(* Schneider Machine Expert - Basic project FlandersHVL, file version 1.8.0.0 *)
(* ProjectInformations: Name=New project *)

HARDWARE
  Cpu 0: TM221CE24R
  ModuleExtensionObject 0: TM3AQ4/G
  ModuleExtensionObject 1: TM2DDO8TT
  ModuleExtensionObject 2: TM2DDO8TT
  EthernetConfiguration: NetworkName=M221, IpAllocationMode=FixedAddress, IpAddress=192.168.1.11, SubnetMask=255.255.255.0
  SerialLineConfiguration: Baud=Baud19200, Parity=ParityEven, DataBits=DataBits8, StopBits=StopBits1, PhysicalMedium=PhysicalMediumRs485, TransmissionMode=TransmissionModeModbusRtu, SlaveId=1, Addressing=SlaveAddressing
  MastTask: UsePeriodScanMode=false, PeriodScan=100
  FastTask: Period=255
  CpuBehavior: StartingMode=StartAsPreviousState, AutoSaveRamOnEeprom=true, WatchdogPeriod=250

SYMBOLS  (address, symbol, comment, settings)
  %M0       STOP
  %M1       RUN_STRIP_PULL_CYCLE
  %M2       EXTEND_CLAMP
  %M3       GLUE_TIMER_DN
  %M4       RUN_GLUE_CYCLE
  %M5       SYSTEM_RUNNING
  %M6       MCR  "Master Control Relay"
  %M7       SYSTEM_IDLE
  %M8       SYSTEM_START
  %M9       PHYSICAL_ALARM_TIMEOUT
  %M10      SYNC_STRIPS
  %M11      ONE_MIN_PASSED
  %M12      NEXT_SPEED
  %M13      START_RPM_TEST
  %M14      STRIP_PULL_STEP_1
  %M15      STRIP_PULL_LAST_STEP
  %M16      SYNC_VACS
  %M17      SYNC_STRIP_CYL_OUT
  %M18      SYN_STRIP_CYL_IN
  %M19      SYNC_PINS
  %M20      SYNC_GLUE
  %M21      SYNC_STRIP_MOTORS
  %M22      TEST_GLUE_RUNNING
  %M23      SLOW_JOG
  %M24      RUN_STRIP_PULL_A_CYCLE
  %M25      STRIP_PULL_A_MANUAL
  %M26      STRIP_PULL_B_MANUAL
  %M27      RUN_STRIP_PULL_B_CYCLE
  %M100     TEST_BIT
  %MW4      DRIVE_MOTOR_SETPOINT
  %MW5      MEDIA_DETECT_SETPOINT
  %MW6      GLUE_A_TOP_ON_DELAY_SETPOINT
  %MW7      VAC_ON_DELAY_SETPOINT
  %MW8      VAC_OFF_DELAY_SETPOINT
  %MW9      PIN_TIMER_SETPOINT
  %MW10     GLUE_A_TOP_OFF_DELAY_SETPOINT
  %MW11     GLUE_A_BOT_ON_DELAY_SETPOINT
  %MW12     GLUE_A_BOT_OFF_DELAY_SETPOINT
  %MW13     GLUE_B_TOP_ON_DELAY_SETPOINT
  %MW14     GLUE_B_TOP_OFF_DELAY_SETPOINT
  %MW15     GLUE_B_BOT_ON_DELAY_SETPOINT
  %MW16     GLUE_B_BOT_OFF_DELAY_SETPOINT
  %MF2      FILTERS_PER_MINUTE
  %TM0      GLUE_A_TOP_ON_DELAY  [Preset=200, Base=TenMilliSeconds]
  %TM1      GLUE_A_TOP_OFF_DELAY  [Preset=70, Base=TenMilliSeconds]
  %TM2      FPM_SPEED_TIMER  [Base=TenMilliSeconds]
  %TM3      MEDIA_DETECT_A_TIMER  [Preset=2000, Base=OneMilliSeconds]
  %TM4      VAC_A_ON_DELAY  [Preset=200, Base=OneMilliSeconds]
  %TM5      VAC_A_OFF_DELAY  [Preset=100, Base=OneMilliSeconds]
  %TM6      PIN_TIMER  [Preset=2, Base=TenMilliSeconds]
  %TM7      GLUE_A_BOT_ON_DELAY  [Base=TenMilliSeconds]
  %TM8      GLUE_A_BOT_OFF_DELAY  [Base=TenMilliSeconds]
  %TM9      GLUE_B_TOP_ON_DELAY  [Base=TenMilliSeconds]
  %TM10     GLUE_B_TOP_OFF_DELAY  [Base=TenMilliSeconds]
  %TM11     GLUE_B_BOT_ON_DELAY  [Base=TenMilliSeconds]
  %TM12     GLUE_B_BOT_OFF_DELAY  [Base=TenMilliSeconds]
  %TM13     VAC_B_ON_DELAY
  %TM14     VAC_B_OFF_DELAY
  %TM15     MEDIA_DETECT_B_TIMER
  %C0       FILTER_PER_MINUTE_COUNTER
  %I0.0     SPEED_DETECT
  %I0.1     FLIGHT_DETECT
  %I0.2     STRIP_CYL_A_OUT
  %I0.3     STRIP_CYL_A_IN
  %I0.4     STRIP_CYL_B_OUT
  %I0.5     STRIP_CYL_B_IN
  %I0.6     MEDIA_DETECT
  %I0.7     STRIP_DETECT_A
  %I0.8     STRIP_DETECT_B
  %I0.9     GLUE_EYE
  %I0.10    SAFETY
  %Q0.0     VAC_A
  %Q0.1     VAC_B
  %Q0.2     STRIP_ARM_A
  %Q0.3     STRIP_ARM_B
  %Q0.4     PIN_A
  %Q0.5     PIN_B
  %Q0.6     GLUE_HEAD_A_TOP
  %Q0.7     GLUE_HEAD_A_BOT
  %Q0.8     GLUE_HEAD_B_TOP
  %Q0.9     GLUE_HEAD_B_BOT
  %QW1.0    DRIVE_MOTOR  [Type=Type_0_10V, Scope=Scope_Customized, Minimum=0, Maximum=7000]
  %Q2.0     PHYSICAL_ALARM
  %Q2.3     PINCH_ROLLER_MOTOR
  %Q2.4     STRIP_B_MOTOR
  %Q2.5     STRIP_A_MOTOR
  %Q2.7     DRIVE_MOTOR_RUN
  %Q3.0     PAD_CUT

POU Strip_Machine_A
  (* SectionNumber=1 *)

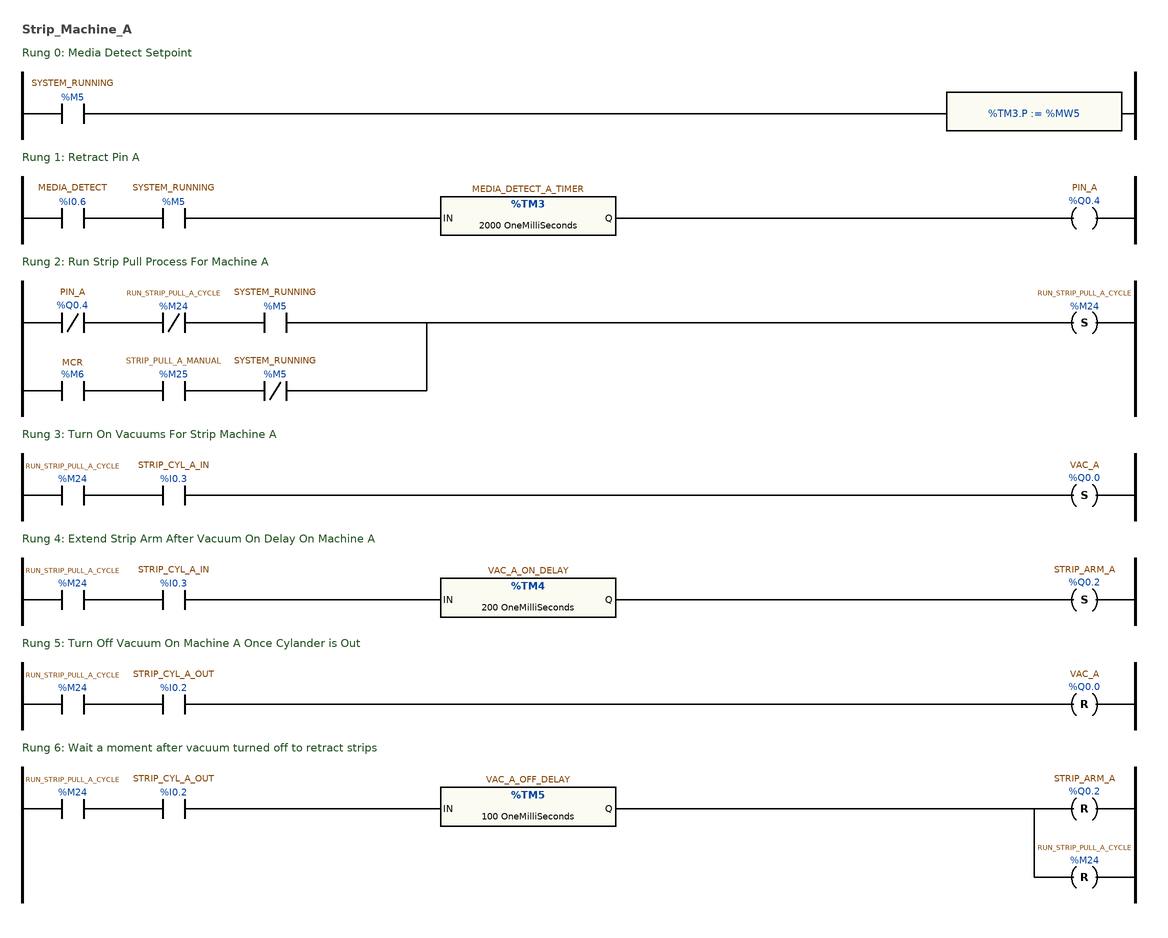

// Rung 0: Media Detect Setpoint
  LD %M5                  (* SYSTEM_RUNNING *)
  [ %TM3.P := %MW5 ]      (* MEDIA_DETECT_A_TIMER, MEDIA_DETECT_SETPOINT *)
  // as ST:
  //   IF SYSTEM_RUNNING THEN MEDIA_DETECT_A_TIMER.P := MEDIA_DETECT_SETPOINT; END_IF;

// Rung 1: Retract Pin A
  BLK %TM3                (* MEDIA_DETECT_A_TIMER *)
  LD %I0.6                (* MEDIA_DETECT *)
  AND %M5                 (* SYSTEM_RUNNING *)
  IN
  OUT_BLK
  LD Q
  ST %Q0.4                (* PIN_A *)
  END_BLK
  // as ST:
  //   MEDIA_DETECT_A_TIMER(IN := MEDIA_DETECT AND SYSTEM_RUNNING);
  //   PIN_A := MEDIA_DETECT_A_TIMER.Q;

// Rung 2: Run Strip Pull Process For Machine A
  LDN %Q0.4               (* PIN_A *)
  ANDN %M24               (* RUN_STRIP_PULL_A_CYCLE *)
  AND %M5                 (* SYSTEM_RUNNING *)
  OR( %M6                 (* MCR *)
  AND %M25                (* STRIP_PULL_A_MANUAL *)
  ANDN %M5                (* SYSTEM_RUNNING *)
  )
  S %M24                  (* RUN_STRIP_PULL_A_CYCLE *)
  // as ST:
  //   IF NOT PIN_A AND NOT RUN_STRIP_PULL_A_CYCLE AND SYSTEM_RUNNING OR MCR AND STRIP_PULL_A_MANUAL AND NOT SYSTEM_RUNNING THEN RUN_STRIP_PULL_A_CYCLE := TRUE; END_IF;

// Rung 3: Turn On Vacuums For Strip Machine A
  LD %M24                 (* RUN_STRIP_PULL_A_CYCLE *)
  AND %I0.3               (* STRIP_CYL_A_IN *)
  S %Q0.0                 (* VAC_A *)
  // as ST:
  //   IF RUN_STRIP_PULL_A_CYCLE AND STRIP_CYL_A_IN THEN VAC_A := TRUE; END_IF;

// Rung 4: Extend Strip Arm After Vacuum On Delay On Machine A
  BLK %TM4                (* VAC_A_ON_DELAY *)
  LD %M24                 (* RUN_STRIP_PULL_A_CYCLE *)
  AND %I0.3               (* STRIP_CYL_A_IN *)
  IN
  OUT_BLK
  LD Q
  S %Q0.2                 (* STRIP_ARM_A *)
  END_BLK
  // as ST:
  //   VAC_A_ON_DELAY(IN := RUN_STRIP_PULL_A_CYCLE AND STRIP_CYL_A_IN);
  //   IF VAC_A_ON_DELAY.Q THEN STRIP_ARM_A := TRUE; END_IF;

// Rung 5: Turn Off Vacuum On Machine A Once Cylander is Out
  LD %M24                 (* RUN_STRIP_PULL_A_CYCLE *)
  AND %I0.2               (* STRIP_CYL_A_OUT *)
  R %Q0.0                 (* VAC_A *)
  // as ST:
  //   IF RUN_STRIP_PULL_A_CYCLE AND STRIP_CYL_A_OUT THEN VAC_A := FALSE; END_IF;

// Rung 6: Wait a moment after vacuum turned off to retract strips
  BLK %TM5                (* VAC_A_OFF_DELAY *)
  LD %M24                 (* RUN_STRIP_PULL_A_CYCLE *)
  AND %I0.2               (* STRIP_CYL_A_OUT *)
  IN
  OUT_BLK
  LD Q
  R %Q0.2                 (* STRIP_ARM_A *)
  R %M24                  (* RUN_STRIP_PULL_A_CYCLE *)
  END_BLK
  // as ST:
  //   VAC_A_OFF_DELAY(IN := RUN_STRIP_PULL_A_CYCLE AND STRIP_CYL_A_OUT);
  //   IF VAC_A_OFF_DELAY.Q THEN STRIP_ARM_A := FALSE; END_IF;
  //   IF VAC_A_OFF_DELAY.Q THEN RUN_STRIP_PULL_A_CYCLE := FALSE; END_IF;

POU High_Power_Devices
  (* SectionNumber=2 *)

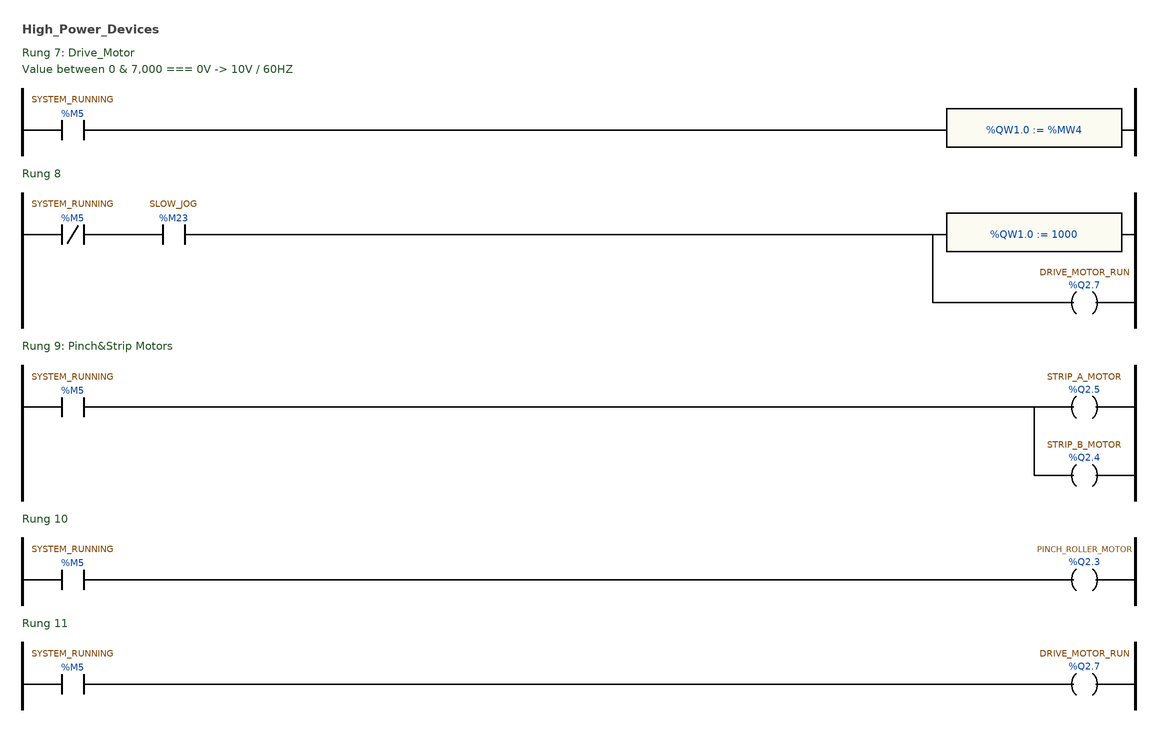

// Rung 7: Drive_Motor
// Value between 0 & 7,000 === 0V -> 10V / 60HZ
  LD %M5                  (* SYSTEM_RUNNING *)
  [ %QW1.0 := %MW4 ]      (* DRIVE_MOTOR, DRIVE_MOTOR_SETPOINT *)
  // as ST:
  //   IF SYSTEM_RUNNING THEN DRIVE_MOTOR := DRIVE_MOTOR_SETPOINT; END_IF;

// Rung 8
  LDN %M5                 (* SYSTEM_RUNNING *)
  AND %M23                (* SLOW_JOG *)
  [ %QW1.0 := 1000 ]      (* DRIVE_MOTOR *)
  ST %Q2.7                (* DRIVE_MOTOR_RUN *)
  // as ST:
  //   IF NOT SYSTEM_RUNNING AND SLOW_JOG THEN DRIVE_MOTOR := 1000; END_IF;
  //   DRIVE_MOTOR_RUN := NOT SYSTEM_RUNNING AND SLOW_JOG;

// Rung 9: Pinch&Strip Motors
  LD %M5                  (* SYSTEM_RUNNING *)
  ST %Q2.5                (* STRIP_A_MOTOR *)
  ST %Q2.4                (* STRIP_B_MOTOR *)
  // as ST:
  //   STRIP_A_MOTOR := SYSTEM_RUNNING;
  //   STRIP_B_MOTOR := SYSTEM_RUNNING;

// Rung 10
  LD %M5                  (* SYSTEM_RUNNING *)
  ST %Q2.3                (* PINCH_ROLLER_MOTOR *)
  // as ST:
  //   PINCH_ROLLER_MOTOR := SYSTEM_RUNNING;

// Rung 11
  LD %M5                  (* SYSTEM_RUNNING *)
  ST %Q2.7                (* DRIVE_MOTOR_RUN *)
  // as ST:
  //   DRIVE_MOTOR_RUN := SYSTEM_RUNNING;

POU RPM
  (* SectionNumber=3 *)

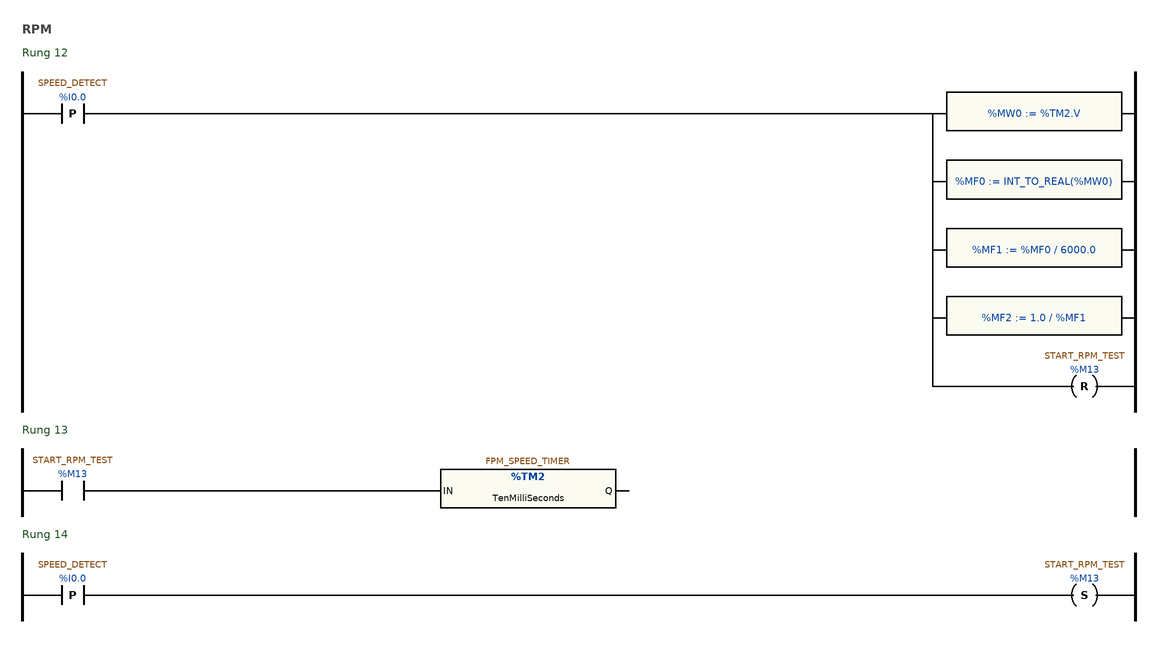

// Rung 12
  LDR %I0.0               (* SPEED_DETECT *)
  [ %MW0 := %TM2.V ]      (* FPM_SPEED_TIMER *)
  [ %MF0 := INT_TO_REAL ( %MW0 ) ]
  [ %MF1 := %MF0 / 6000.0 ]
  [ %MF2 := 1.0 / %MF1 ]  (* FILTERS_PER_MINUTE *)
  R %M13                  (* START_RPM_TEST *)
  // as ST:
  //   IF RISING(SPEED_DETECT) THEN %MW0 := FPM_SPEED_TIMER.V; END_IF;
  //   IF RISING(SPEED_DETECT) THEN %MF0 := INT_TO_REAL ( %MW0 ); END_IF;
  //   IF RISING(SPEED_DETECT) THEN %MF1 := %MF0  /  6000.0; END_IF;
  //   IF RISING(SPEED_DETECT) THEN FILTERS_PER_MINUTE := 1.0  /  %MF1; END_IF;
  //   IF RISING(SPEED_DETECT) THEN START_RPM_TEST := FALSE; END_IF;

// Rung 13
  BLK %TM2                (* FPM_SPEED_TIMER *)
  LD %M13                 (* START_RPM_TEST *)
  IN
  END_BLK
  // as ST:
  //   FPM_SPEED_TIMER(IN := START_RPM_TEST);

// Rung 14
  LDR %I0.0               (* SPEED_DETECT *)
  S %M13                  (* START_RPM_TEST *)
  // as ST:
  //   IF RISING(SPEED_DETECT) THEN START_RPM_TEST := TRUE; END_IF;

POU Synchronize
  (* SectionNumber=4 *)

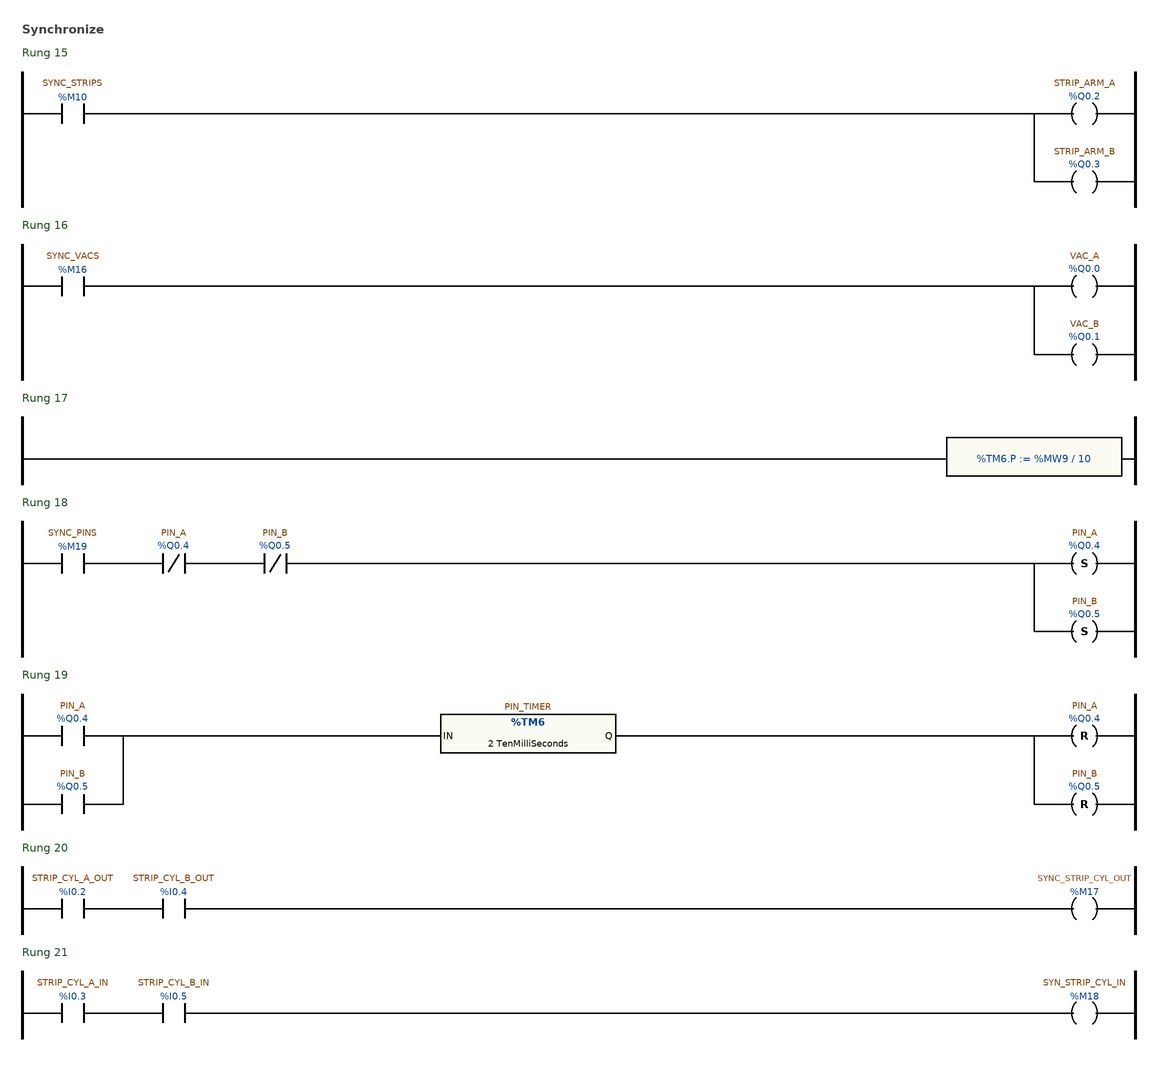

// Rung 15
  LD %M10                 (* SYNC_STRIPS *)
  ST %Q0.2                (* STRIP_ARM_A *)
  ST %Q0.3                (* STRIP_ARM_B *)
  // as ST:
  //   STRIP_ARM_A := SYNC_STRIPS;
  //   STRIP_ARM_B := SYNC_STRIPS;

// Rung 16
  LD %M16                 (* SYNC_VACS *)
  ST %Q0.0                (* VAC_A *)
  ST %Q0.1                (* VAC_B *)
  // as ST:
  //   VAC_A := SYNC_VACS;
  //   VAC_B := SYNC_VACS;

// Rung 17
  LD 1
  [ %TM6.P := %MW9 / 10 ] (* PIN_TIMER, PIN_TIMER_SETPOINT *)
  // as ST:
  //   PIN_TIMER.P := PIN_TIMER_SETPOINT / 10;

// Rung 18
  LD %M19                 (* SYNC_PINS *)
  ANDN %Q0.4              (* PIN_A *)
  ANDN %Q0.5              (* PIN_B *)
  S %Q0.4                 (* PIN_A *)
  S %Q0.5                 (* PIN_B *)
  // as ST:
  //   _t1 := SYNC_PINS AND NOT PIN_A AND NOT PIN_B;
  //   IF _t1 THEN PIN_A := TRUE; END_IF;
  //   IF _t1 THEN PIN_B := TRUE; END_IF;

// Rung 19
  BLK %TM6                (* PIN_TIMER *)
  LD %Q0.4                (* PIN_A *)
  OR %Q0.5                (* PIN_B *)
  IN
  OUT_BLK
  LD Q
  R %Q0.4                 (* PIN_A *)
  R %Q0.5                 (* PIN_B *)
  END_BLK
  // as ST:
  //   PIN_TIMER(IN := PIN_A OR PIN_B);
  //   IF PIN_TIMER.Q THEN PIN_A := FALSE; END_IF;
  //   IF PIN_TIMER.Q THEN PIN_B := FALSE; END_IF;

// Rung 20
  LD %I0.2                (* STRIP_CYL_A_OUT *)
  AND %I0.4               (* STRIP_CYL_B_OUT *)
  ST %M17                 (* SYNC_STRIP_CYL_OUT *)
  // as ST:
  //   SYNC_STRIP_CYL_OUT := STRIP_CYL_A_OUT AND STRIP_CYL_B_OUT;

// Rung 21
  LD %I0.3                (* STRIP_CYL_A_IN *)
  AND %I0.5               (* STRIP_CYL_B_IN *)
  ST %M18                 (* SYN_STRIP_CYL_IN *)
  // as ST:
  //   SYN_STRIP_CYL_IN := STRIP_CYL_A_IN AND STRIP_CYL_B_IN;

POU Sytem Signals
  (* SectionNumber=5 *)

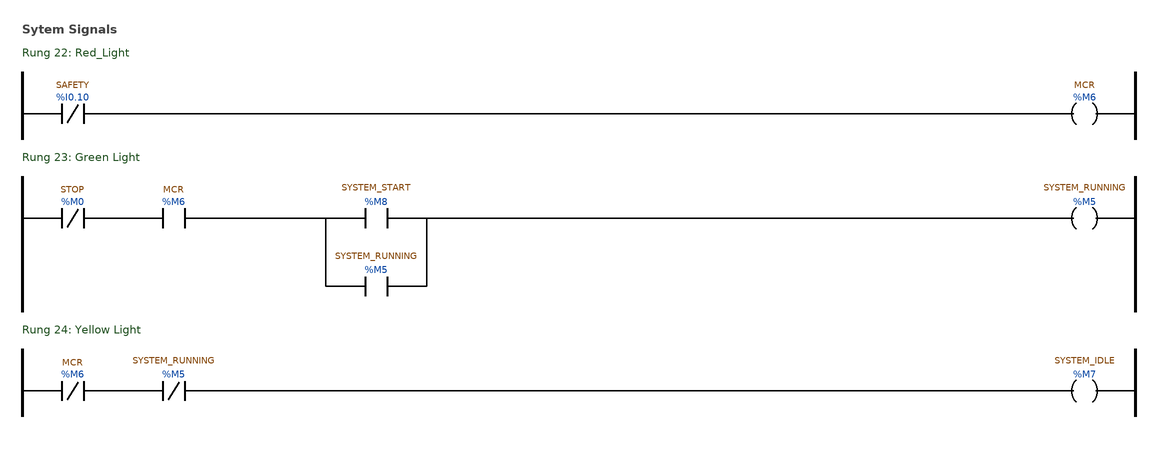

// Rung 22: Red_Light
  LDN %I0.10              (* SAFETY *)
  ST %M6                  (* MCR *)
  // as ST:
  //   MCR := NOT SAFETY;

// Rung 23: Green Light
  LDN %M0                 (* STOP *)
  AND %M6                 (* MCR *)
  AND( %M8                (* SYSTEM_START *)
  OR %M5                  (* SYSTEM_RUNNING *)
  )
  ST %M5                  (* SYSTEM_RUNNING *)
  // as ST:
  //   SYSTEM_RUNNING := NOT STOP AND MCR AND (SYSTEM_START OR SYSTEM_RUNNING);

// Rung 24: Yellow Light
  LDN %M6                 (* MCR *)
  ANDN %M5                (* SYSTEM_RUNNING *)
  ST %M7                  (* SYSTEM_IDLE *)
  // as ST:
  //   SYSTEM_IDLE := NOT MCR AND NOT SYSTEM_RUNNING;

POU Glue
  (* SectionNumber=6 *)

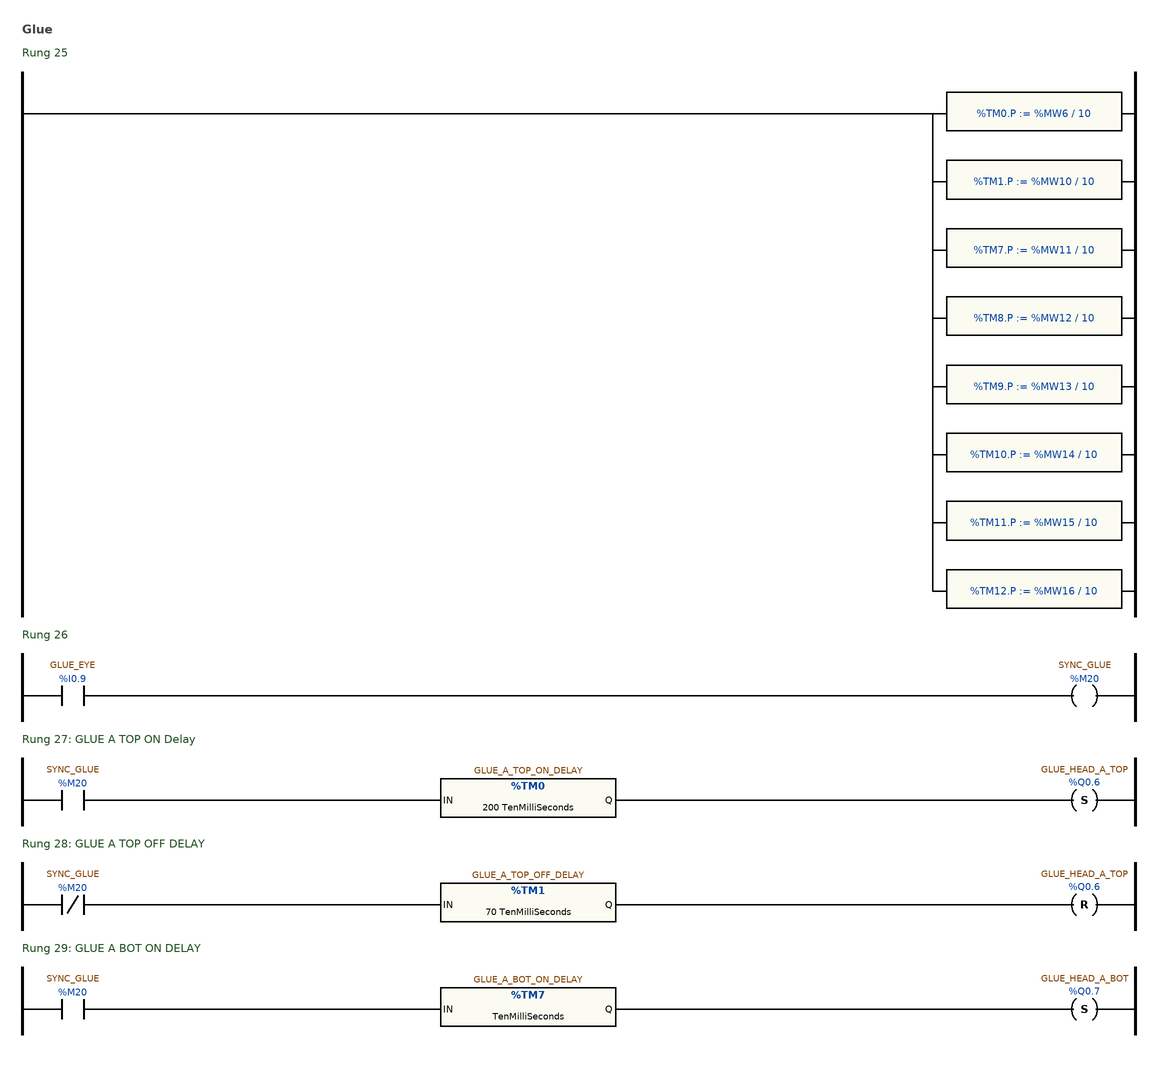

// Rung 25
  LD 1
  [%TM0.P := %MW6 / 10]   (* GLUE_A_TOP_ON_DELAY, GLUE_A_TOP_ON_DELAY_SETPOINT *)
  [%TM1.P := %MW10 / 10]  (* GLUE_A_TOP_OFF_DELAY, GLUE_A_TOP_OFF_DELAY_SETPOINT *)
  [%TM7.P := %MW11 / 10]  (* GLUE_A_BOT_ON_DELAY, GLUE_A_BOT_ON_DELAY_SETPOINT *)
  [%TM8.P := %MW12 / 10]  (* GLUE_A_BOT_OFF_DELAY, GLUE_A_BOT_OFF_DELAY_SETPOINT *)
  [%TM9.P := %MW13 / 10]  (* GLUE_B_TOP_ON_DELAY, GLUE_B_TOP_ON_DELAY_SETPOINT *)
  [%TM10.P := %MW14 / 10] (* GLUE_B_TOP_OFF_DELAY, GLUE_B_TOP_OFF_DELAY_SETPOINT *)
  [%TM11.P := %MW15 / 10] (* GLUE_B_BOT_ON_DELAY, GLUE_B_BOT_ON_DELAY_SETPOINT *)
  [%TM12.P := %MW16 / 10] (* GLUE_B_BOT_OFF_DELAY, GLUE_B_BOT_OFF_DELAY_SETPOINT *)
  // as ST:
  //   GLUE_A_TOP_ON_DELAY.P := GLUE_A_TOP_ON_DELAY_SETPOINT / 10;
  //   GLUE_A_TOP_OFF_DELAY.P := GLUE_A_TOP_OFF_DELAY_SETPOINT / 10;
  //   GLUE_A_BOT_ON_DELAY.P := GLUE_A_BOT_ON_DELAY_SETPOINT / 10;
  //   GLUE_A_BOT_OFF_DELAY.P := GLUE_A_BOT_OFF_DELAY_SETPOINT / 10;
  //   GLUE_B_TOP_ON_DELAY.P := GLUE_B_TOP_ON_DELAY_SETPOINT / 10;
  //   GLUE_B_TOP_OFF_DELAY.P := GLUE_B_TOP_OFF_DELAY_SETPOINT / 10;
  //   GLUE_B_BOT_ON_DELAY.P := GLUE_B_BOT_ON_DELAY_SETPOINT / 10;
  //   GLUE_B_BOT_OFF_DELAY.P := GLUE_B_BOT_OFF_DELAY_SETPOINT / 10;

// Rung 26
  LD %I0.9                (* GLUE_EYE *)
  ST %M20                 (* SYNC_GLUE *)
  // as ST:
  //   SYNC_GLUE := GLUE_EYE;

// Rung 27: GLUE A TOP ON Delay
  BLK %TM0                (* GLUE_A_TOP_ON_DELAY *)
  LD %M20                 (* SYNC_GLUE *)
  IN
  OUT_BLK
  LD Q
  S %Q0.6                 (* GLUE_HEAD_A_TOP *)
  END_BLK
  // as ST:
  //   GLUE_A_TOP_ON_DELAY(IN := SYNC_GLUE);
  //   IF GLUE_A_TOP_ON_DELAY.Q THEN GLUE_HEAD_A_TOP := TRUE; END_IF;

// Rung 28: GLUE A TOP OFF DELAY
  BLK %TM1                (* GLUE_A_TOP_OFF_DELAY *)
  LDN %M20                (* SYNC_GLUE *)
  IN
  OUT_BLK
  LD Q
  R %Q0.6                 (* GLUE_HEAD_A_TOP *)
  END_BLK
  // as ST:
  //   GLUE_A_TOP_OFF_DELAY(IN := NOT SYNC_GLUE);
  //   IF GLUE_A_TOP_OFF_DELAY.Q THEN GLUE_HEAD_A_TOP := FALSE; END_IF;

// Rung 29: GLUE A BOT ON DELAY
  BLK %TM7                (* GLUE_A_BOT_ON_DELAY *)
  LD %M20                 (* SYNC_GLUE *)
  IN
  OUT_BLK
  LD Q
  S %Q0.7                 (* GLUE_HEAD_A_BOT *)
  END_BLK
  // as ST:
  //   GLUE_A_BOT_ON_DELAY(IN := SYNC_GLUE);
  //   IF GLUE_A_BOT_ON_DELAY.Q THEN GLUE_HEAD_A_BOT := TRUE; END_IF;

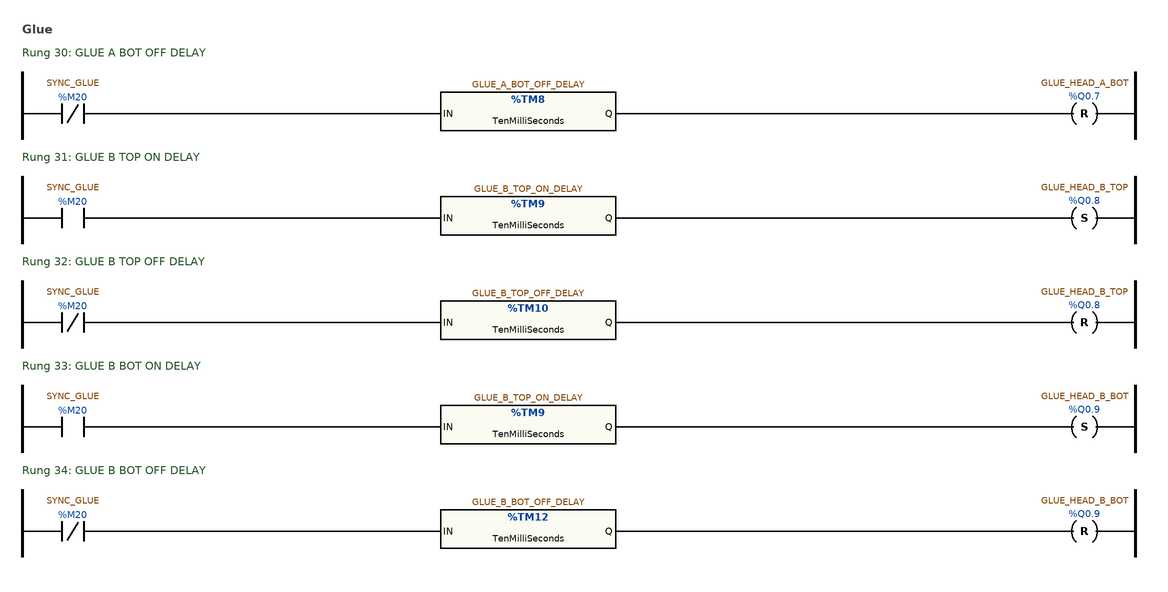

// Rung 30: GLUE A BOT OFF DELAY
  BLK %TM8                (* GLUE_A_BOT_OFF_DELAY *)
  LDN %M20                (* SYNC_GLUE *)
  IN
  OUT_BLK
  LD Q
  R %Q0.7                 (* GLUE_HEAD_A_BOT *)
  END_BLK
  // as ST:
  //   GLUE_A_BOT_OFF_DELAY(IN := NOT SYNC_GLUE);
  //   IF GLUE_A_BOT_OFF_DELAY.Q THEN GLUE_HEAD_A_BOT := FALSE; END_IF;

// Rung 31: GLUE B TOP ON DELAY
  BLK %TM9                (* GLUE_B_TOP_ON_DELAY *)
  LD %M20                 (* SYNC_GLUE *)
  IN
  OUT_BLK
  LD Q
  S %Q0.8                 (* GLUE_HEAD_B_TOP *)
  END_BLK
  // as ST:
  //   GLUE_B_TOP_ON_DELAY(IN := SYNC_GLUE);
  //   IF GLUE_B_TOP_ON_DELAY.Q THEN GLUE_HEAD_B_TOP := TRUE; END_IF;

// Rung 32: GLUE B TOP OFF DELAY
  BLK %TM10               (* GLUE_B_TOP_OFF_DELAY *)
  LDN %M20                (* SYNC_GLUE *)
  IN
  OUT_BLK
  LD Q
  R %Q0.8                 (* GLUE_HEAD_B_TOP *)
  END_BLK
  // as ST:
  //   GLUE_B_TOP_OFF_DELAY(IN := NOT SYNC_GLUE);
  //   IF GLUE_B_TOP_OFF_DELAY.Q THEN GLUE_HEAD_B_TOP := FALSE; END_IF;

// Rung 33: GLUE B BOT ON DELAY
  BLK %TM9                (* GLUE_B_TOP_ON_DELAY *)
  LD %M20                 (* SYNC_GLUE *)
  IN
  OUT_BLK
  LD Q
  S %Q0.9                 (* GLUE_HEAD_B_BOT *)
  END_BLK
  // as ST:
  //   GLUE_B_TOP_ON_DELAY(IN := SYNC_GLUE);
  //   IF GLUE_B_TOP_ON_DELAY.Q THEN GLUE_HEAD_B_BOT := TRUE; END_IF;

// Rung 34: GLUE B BOT OFF DELAY
  BLK %TM12               (* GLUE_B_BOT_OFF_DELAY *)
  LDN %M20                (* SYNC_GLUE *)
  IN
  OUT_BLK
  LD Q
  R %Q0.9                 (* GLUE_HEAD_B_BOT *)
  END_BLK
  // as ST:
  //   GLUE_B_BOT_OFF_DELAY(IN := NOT SYNC_GLUE);
  //   IF GLUE_B_BOT_OFF_DELAY.Q THEN GLUE_HEAD_B_BOT := FALSE; END_IF;

POU Timer_Setpoints
  (* SectionNumber=7 *)

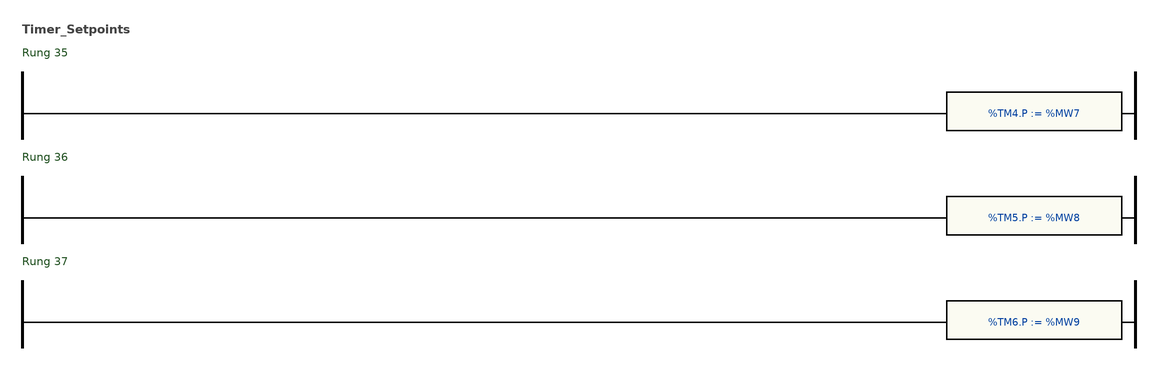

// Rung 35
  LD 1
  [ %TM4.P := %MW7 ]      (* VAC_A_ON_DELAY, VAC_ON_DELAY_SETPOINT *)
  // as ST:
  //   VAC_A_ON_DELAY.P := VAC_ON_DELAY_SETPOINT;

// Rung 36
  LD 1
  [ %TM5.P := %MW8 ]      (* VAC_A_OFF_DELAY, VAC_OFF_DELAY_SETPOINT *)
  // as ST:
  //   VAC_A_OFF_DELAY.P := VAC_OFF_DELAY_SETPOINT;

// Rung 37
  LD 1
  [ %TM6.P := %MW9 ]      (* PIN_TIMER, PIN_TIMER_SETPOINT *)
  // as ST:
  //   PIN_TIMER.P := PIN_TIMER_SETPOINT;

POU Pad Cutter
  (* SectionNumber=0 *)

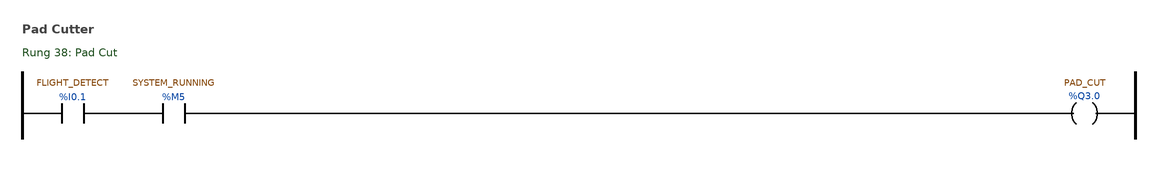

// Rung 38: Pad Cut
  LD %I0.1                (* FLIGHT_DETECT *)
  AND %M5                 (* SYSTEM_RUNNING *)
  ST %Q3.0                (* PAD_CUT *)
  // as ST:
  //   PAD_CUT := FLIGHT_DETECT AND SYSTEM_RUNNING;

POU Strip_Machine_B
  (* SectionNumber=1 *)

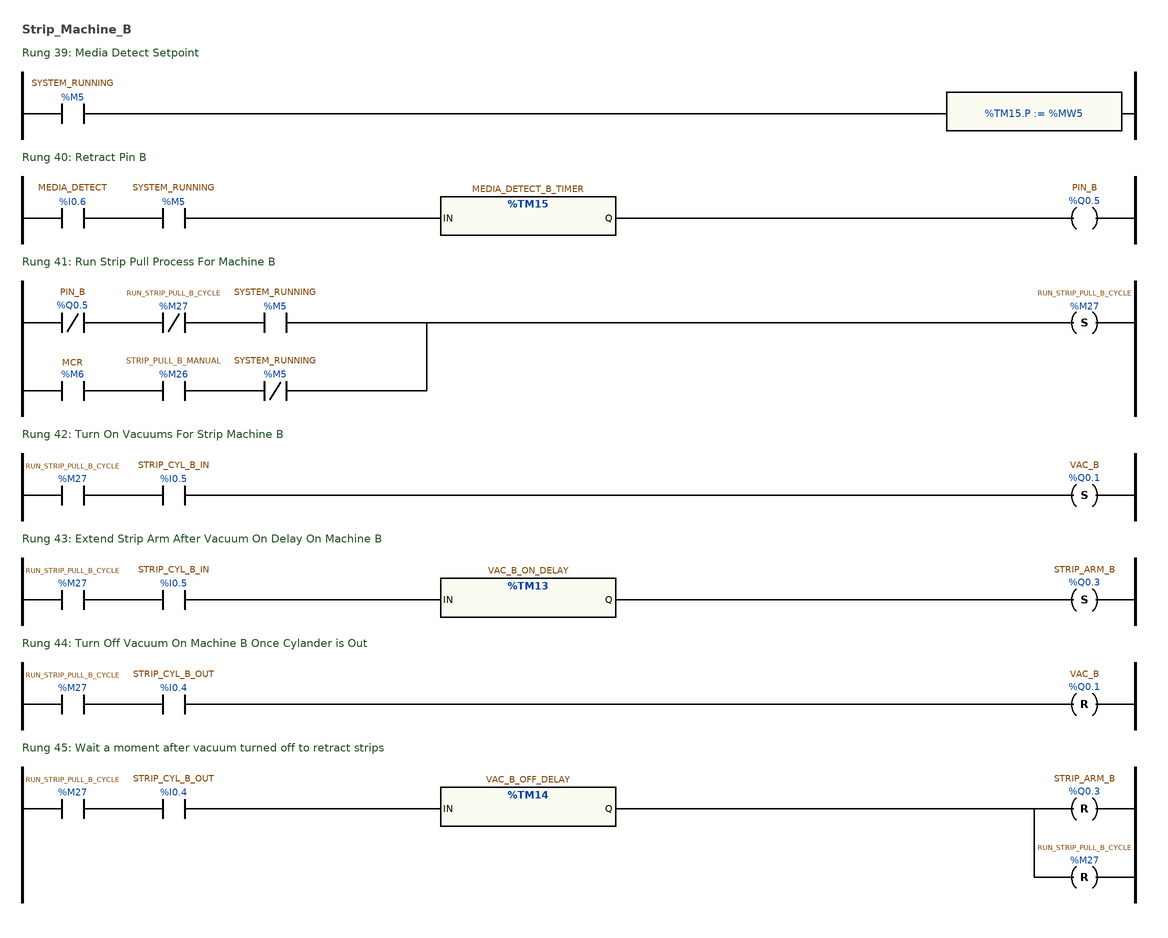

// Rung 39: Media Detect Setpoint
  LD %M5                  (* SYSTEM_RUNNING *)
  [ %TM15.P := %MW5 ]     (* MEDIA_DETECT_B_TIMER, MEDIA_DETECT_SETPOINT *)
  // as ST:
  //   IF SYSTEM_RUNNING THEN MEDIA_DETECT_B_TIMER.P := MEDIA_DETECT_SETPOINT; END_IF;

// Rung 40: Retract Pin B
  BLK %TM15               (* MEDIA_DETECT_B_TIMER *)
  LD %I0.6                (* MEDIA_DETECT *)
  AND %M5                 (* SYSTEM_RUNNING *)
  IN
  OUT_BLK
  LD Q
  ST %Q0.5                (* PIN_B *)
  END_BLK
  // as ST:
  //   MEDIA_DETECT_B_TIMER(IN := MEDIA_DETECT AND SYSTEM_RUNNING);
  //   PIN_B := MEDIA_DETECT_B_TIMER.Q;

// Rung 41: Run Strip Pull Process For Machine B
  LDN %Q0.5               (* PIN_B *)
  ANDN %M27               (* RUN_STRIP_PULL_B_CYCLE *)
  AND %M5                 (* SYSTEM_RUNNING *)
  OR( %M6                 (* MCR *)
  AND %M26                (* STRIP_PULL_B_MANUAL *)
  ANDN %M5                (* SYSTEM_RUNNING *)
  )
  S %M27                  (* RUN_STRIP_PULL_B_CYCLE *)
  // as ST:
  //   IF NOT PIN_B AND NOT RUN_STRIP_PULL_B_CYCLE AND SYSTEM_RUNNING OR MCR AND STRIP_PULL_B_MANUAL AND NOT SYSTEM_RUNNING THEN RUN_STRIP_PULL_B_CYCLE := TRUE; END_IF;

// Rung 42: Turn On Vacuums For Strip Machine B
  LD %M27                 (* RUN_STRIP_PULL_B_CYCLE *)
  AND %I0.5               (* STRIP_CYL_B_IN *)
  S %Q0.1                 (* VAC_B *)
  // as ST:
  //   IF RUN_STRIP_PULL_B_CYCLE AND STRIP_CYL_B_IN THEN VAC_B := TRUE; END_IF;

// Rung 43: Extend Strip Arm After Vacuum On Delay On Machine B
  BLK %TM13               (* VAC_B_ON_DELAY *)
  LD %M27                 (* RUN_STRIP_PULL_B_CYCLE *)
  AND %I0.5               (* STRIP_CYL_B_IN *)
  IN
  OUT_BLK
  LD Q
  S %Q0.3                 (* STRIP_ARM_B *)
  END_BLK
  // as ST:
  //   VAC_B_ON_DELAY(IN := RUN_STRIP_PULL_B_CYCLE AND STRIP_CYL_B_IN);
  //   IF VAC_B_ON_DELAY.Q THEN STRIP_ARM_B := TRUE; END_IF;

// Rung 44: Turn Off Vacuum On Machine B Once Cylander is Out
  LD %M27                 (* RUN_STRIP_PULL_B_CYCLE *)
  AND %I0.4               (* STRIP_CYL_B_OUT *)
  R %Q0.1                 (* VAC_B *)
  // as ST:
  //   IF RUN_STRIP_PULL_B_CYCLE AND STRIP_CYL_B_OUT THEN VAC_B := FALSE; END_IF;

// Rung 45: Wait a moment after vacuum turned off to retract strips
  BLK %TM14               (* VAC_B_OFF_DELAY *)
  LD %M27                 (* RUN_STRIP_PULL_B_CYCLE *)
  AND %I0.4               (* STRIP_CYL_B_OUT *)
  IN
  OUT_BLK
  LD Q
  R %Q0.3                 (* STRIP_ARM_B *)
  R %M27                  (* RUN_STRIP_PULL_B_CYCLE *)
  END_BLK
  // as ST:
  //   VAC_B_OFF_DELAY(IN := RUN_STRIP_PULL_B_CYCLE AND STRIP_CYL_B_OUT);
  //   IF VAC_B_OFF_DELAY.Q THEN STRIP_ARM_B := FALSE; END_IF;
  //   IF VAC_B_OFF_DELAY.Q THEN RUN_STRIP_PULL_B_CYCLE := FALSE; END_IF;
